INTERFACE I_MotionInterlocks

PROPERTY AllBackwardEnabled : BOOL
GET
END_GET
END_PROPERTY

PROPERTY AllEnabled : BOOL
GET
END_GET
END_PROPERTY

PROPERTY AllForwardEnabled : BOOL
GET
END_GET
END_PROPERTY

PROPERTY AxisState : MC_AxisStates
SET
END_SET
END_PROPERTY

PROPERTY CmdReset : BOOL
SET
END_SET
END_PROPERTY

PROPERTY Enable : BOOL
GET
END_GET
END_PROPERTY

PROPERTY EnableDone : BOOL
GET
END_GET
END_PROPERTY

PROPERTY EnableMode : E_StageEnableMode
GET
END_GET
SET
END_SET
END_PROPERTY

PROPERTY EPSOk : BOOL
GET
END_GET
SET
END_SET
END_PROPERTY

PROPERTY Error : BOOL
SET
END_SET
END_PROPERTY

PROPERTY Execute : BOOL
GET
END_GET
SET
END_SET
END_PROPERTY

PROPERTY GantryAxis : BOOL
GET
END_GET
SET
END_SET
END_PROPERTY

PROPERTY GantryBackwardEnable : BOOL
GET
END_GET
SET
END_SET
END_PROPERTY

PROPERTY GantryForwardEnable : BOOL
GET
END_GET
SET
END_SET
END_PROPERTY

PROPERTY HardwareEnable : BOOL
GET
END_GET
SET
END_SET
END_PROPERTY

PROPERTY HomingBusy : BOOL
SET
END_SET
END_PROPERTY

PROPERTY InterlockExec : BOOL
GET
END_GET
END_PROPERTY

PROPERTY LimBwdEnable : BOOL
GET
END_GET
SET
END_SET
END_PROPERTY

PROPERTY LimFwdEnable : BOOL
GET
END_GET
SET
END_SET
END_PROPERTY

PROPERTY LimHit : BOOL
GET
END_GET
END_PROPERTY

PROPERTY LimHome : BOOL
GET
END_GET
SET
END_SET
END_PROPERTY

PROPERTY MoveBusy : BOOL
SET
END_SET
END_PROPERTY

PROPERTY MoveDone : BOOL
SET
END_SET
END_PROPERTY

PROPERTY NewMoveReq : BOOL
GET
END_GET
SET
END_SET
END_PROPERTY

PROPERTY PowerSelf : BOOL
GET
END_GET
SET
END_SET
END_PROPERTY

PROPERTY PrepareDisable : BOOL
GET
END_GET
END_PROPERTY

PROPERTY SafetyReady : BOOL
GET
END_GET
SET
END_SET
END_PROPERTY

PROPERTY SoftInterlock : BOOL
GET
END_GET
SET
END_SET
END_PROPERTY

PROPERTY UserEnable : BOOL
GET
END_GET
SET
END_SET
END_PROPERTY

{warning 'Add property implementation'}
PROPERTY WarnID : UINT
GET
END_GET
END_PROPERTY

PROPERTY WarningMsg : STRING
GET
END_GET
END_PROPERTY

END_INTERFACE

(* stored: Version 1.1.0.1
   Itf I_MotionInterlocks: Id {7ac89254-d732-4980-b014-871a72f21fa7}
   Property AllBackwardEnabled: Id {44fa7548-c01f-4da3-a333-2275934d3112}
   Get Get: Id {8e243d13-164d-4d5d-8112-387f3a8b0fca}
   Property AllEnabled: Id {4d69c415-64ae-45e5-8741-9ee750fa41cf}
   Get Get: Id {09b8b64d-72b0-467d-b693-fa3e229ceb18}
   Property AllForwardEnabled: Id {3ce5ac2e-1c09-4fd1-941c-2cbe06026596}
   Get Get: Id {8ac731aa-4431-4ad2-aad0-76448e67d881}
   Property AxisState: Id {d5bc9801-34cb-48bc-9948-9b462c881460}
   Set Set: Id {7ec24f46-e413-461c-bd66-db5b0cbe9b35}
   Property CmdReset: Id {2b172bef-4c6d-4101-98cd-66ec53623cad}
   Set Set: Id {2d1bf663-ca00-4ccd-b8e7-f23b19c37b45}
   Property Enable: Id {ea046e47-fac5-4980-8551-1d79603777cd}
   Get Get: Id {a3a0e76d-a288-4b3d-aec5-a7603eaf4218}
   Property EnableDone: Id {f2d2f74b-7415-4ea0-8340-cc5a7fb4c649}
   Get Get: Id {2a482f56-07c2-47eb-b118-051cd2b9d33a}
   Property EnableMode: Id {67601fde-f3ba-4ea2-8dbf-89942a2b645f}
   Get Get: Id {676864db-ffb0-4c69-975c-03ab7e9f4fb5}
   Set Set: Id {095f7675-4fda-466c-b0d4-7e5b6e751e78}
   Property EPSOk: Id {2ab43de3-0abf-4f29-b1d9-776886efae5d}
   Get Get: Id {963baa30-2ed7-4807-8ba8-e09808456204}
   Set Set: Id {8bc5bd75-07a7-44de-ac8f-1ad8ff551029}
   Property Error: Id {6f5e8df3-6a99-431a-85cd-5900de0cb2ed}
   Set Set: Id {457b72ab-c009-40bc-a96e-195ff378bbbf}
   Property Execute: Id {d053da7d-cd84-4d5e-bc3e-1b66a9f9aae1}
   Get Get: Id {5671b1bc-3636-44ea-b7c8-078f8bace32e}
   Set Set: Id {bd9d3d4c-231d-44a1-b80c-a9cf1888b9a9}
   Property GantryAxis: Id {56006ae1-c693-47b5-a7b2-3327681468a5}
   Get Get: Id {29ac787b-548b-40c0-aee0-72e462d082cc}
   Set Set: Id {46c657f3-a086-4fed-b359-12c3fd9d60d1}
   Property GantryBackwardEnable: Id {f904ecbf-7926-4b97-a553-c1e262839afe}
   Get Get: Id {f53ef5a8-39bd-4b60-8938-d7e59932b51a}
   Set Set: Id {a5df2c27-bd1f-4e41-b211-426d9f0beb2c}
   Property GantryForwardEnable: Id {a1dbb698-133c-46e9-819b-17b9b9f21b23}
   Get Get: Id {bd086b46-a9ef-4695-a19b-7f1e76359447}
   Set Set: Id {35f02b45-8b53-4e6a-9812-d446b45c27b1}
   Property HardwareEnable: Id {855c6e4b-bfed-49b3-bdec-eafa65093aa9}
   Get Get: Id {3bc8c738-8360-4ae7-9ad5-cf8bc24dacf1}
   Set Set: Id {489a79c4-eb9c-4a2f-baad-54d7878ac34a}
   Property HomingBusy: Id {13c4642a-cce9-4a6b-a728-b39ae7081a30}
   Set Set: Id {489c89f2-7ddf-4c94-9a43-8900bb688f7a}
   Property InterlockExec: Id {99ca9de1-0720-480d-87e8-bfb0d02920c3}
   Get Get: Id {55e84a45-a8fa-4728-9be6-724774efdfb5}
   Property LimBwdEnable: Id {4f071531-664b-43fb-9b98-46ce706701d6}
   Get Get: Id {9187b4a7-a42c-4364-a237-fe27d1b092b0}
   Set Set: Id {b9aff11f-e55e-4ea0-a544-b45c3be44f95}
   Property LimFwdEnable: Id {63378470-96d4-47b7-a381-4d50609bb5a2}
   Get Get: Id {13bb15a4-f20a-4eed-b421-340a7c7204a2}
   Set Set: Id {7ad36303-dc71-4d7a-b996-eaec00eed2df}
   Property LimHit: Id {00f31b83-20b0-4e18-bb57-b84a58adcd1b}
   Get Get: Id {dc48a399-6ef3-4f49-9589-4858181b8029}
   Property LimHome: Id {43b3c4e0-2529-4ca2-94b6-01308791bd0f}
   Get Get: Id {fa4d37b3-5d02-4b73-968e-4a37c39a113f}
   Set Set: Id {aca26340-7624-4f3a-8bc3-b354a8230aaf}
   Property MoveBusy: Id {c47b4aa2-3195-4ba8-b3b3-e05d5f5551d5}
   Set Set: Id {bd5d510c-b0f2-4b6a-b7ab-f43a0869e21a}
   Property MoveDone: Id {4c6f2964-50b7-453e-8868-a73dd4159a2d}
   Set Set: Id {bb507fd3-3547-4579-b7f1-378af88a801c}
   Property NewMoveReq: Id {482dbe2c-aada-46e4-a4b0-e1927f9c0bd2}
   Get Get: Id {4c5cc58e-3e8b-4496-a7da-4d638c7f0868}
   Set Set: Id {fdb42c11-1971-442a-a56c-238729145db3}
   Property PowerSelf: Id {af7539d4-48fa-4915-a716-1585614bb150}
   Get Get: Id {832ea85a-44e1-43f2-84fb-a9a7ce8a9a54}
   Set Set: Id {3ab08d4c-6e93-4a5c-b644-d0f7e3500942}
   Property PrepareDisable: Id {06826ef8-4820-4e0e-99a8-95eabef50bc5}
   Get Get: Id {1218905d-5cb7-4bcc-84f4-3911642dcd18}
   Property SafetyReady: Id {c4a49c88-eac4-4e17-84d8-41063fa69887}
   Get Get: Id {67ae7808-2d1e-4903-92a5-9e496ca319df}
   Set Set: Id {6c96cb36-0d7f-4cc1-9cb5-39659c0eaab3}
   Property SoftInterlock: Id {84b462fb-97b6-4df9-b44c-e4fc3600b4a1}
   Get Get: Id {4c848c4c-616c-4dea-8b19-c0ad93f2399c}
   Set Set: Id {7e455863-b97d-4ef2-8c0a-175169e8ec44}
   Property UserEnable: Id {b04015ea-94bc-4cb0-a1f4-ebb6556cce84}
   Get Get: Id {3936eba9-09b5-408d-b793-738e943f6fd9}
   Set Set: Id {6f48e91f-76ea-4390-901a-a92e460215eb}
   Property WarnID: Id {be859d4c-20b0-48fc-90e8-64961601a870}
   Get Get: Id {aff35a25-4efa-4678-8127-c8619732e505}
   Property WarningMsg: Id {bf7b81d5-c154-46fb-b50d-9188e5c9721a}
   Get Get: Id {904bcd85-b16b-4196-9319-f47b5feeb0d9} *)
